{attribute addProperty BoxType "KL9940-0050"}
{attribute addProperty Id "Channel_1Channel_CB1ECEDB00"}
{attribute addProperty CRC "142024747"}
{attribute addProperty SizeInBites "0"}
{attribute addProperty SizeInBytes "0"}
TYPE KL_0877202B :
STRUCT
	{attribute addProperty Name "Channel_1"}
	Channel_1 : Channel_CB1ECEDB;
END_STRUCT
END_TYPE

(* stored: Version 1.2.0.0, ProductVersion 3.1.4024.9
   DUT KL_0877202B: Id {53ed7530-5206-4a1f-9061-60b5bfd8ff8f} *)
